// TwinCAT 3 PLC project PLC
// Title: abc
// Company: abc
// ProjectVersion: 1.0
// ProgramVersion: 3.1.0.8
// libraries:
//   Tc2_Standard, * (Beckhoff Automation GmbH)
//   Tc2_System, * (Beckhoff Automation GmbH)
//   Tc3_Interfaces, * (Beckhoff Automation GmbH)
//   Tc3_Module, * (Beckhoff Automation GmbH)
// project tree:
//   DUTs/ PLCStruct.TcDUT, TComplexStruct.TcDUT, TSimpleStruct.TcDUT (not stored)
//   GVLs/ GVL.TcGVL
//   / PlcTask.TcTTO (not stored)
//   POUs/ FB_Math.TcPOU, MAIN.TcPOU
//   Version/ Global_Version.TcGVL
// real-time tasks:
//   TASK PlcTask: cycle T#10ms, priority 20, ADS port 350

// ---- DUTs/PLCStruct.TcDUT
TYPE PLCStruct :
STRUCT
	intVal 	: INT;
  	dintVal	: DINT;
  	byteVal	: SINT;
  	lrealVal: LREAL;
  	realVal	: REAL;
END_STRUCT
END_TYPE

// ---- DUTs/TComplexStruct.TcDUT
TYPE TComplexStruct :
STRUCT
	intVal 			: INT:=1200;
	dintArr			: ARRAY[0..3] OF DINT := [1,2,3,4];
	boolVal			: BOOL := FALSE;
	byteVal			: BYTE:=10;
	stringVal 		: STRING(5) := 'hallo';
	simpleStruct1	:  TSimpleStruct;
END_STRUCT
END_TYPE

// ---- GVLs/GVL.TcGVL
VAR_GLOBAL
	//Sample21
	REAL32_1 AT %MB0 : REAL;  (* 1 *)
        REAL32_2 AT %MB4 : REAL;  (* 2 *)
        REAL32_3 AT %MB8 : REAL;  (* 3 *)
        REAL32_4 AT %MB12: REAL;  (* 4 *)
        REAL32_5 AT %MB16: REAL;  (* 5 *)

        REAL64_1 AT %MB20 : LREAL;  (* 6 *)
        REAL64_2 AT %MB28 : LREAL;  (* 7 *)
        REAL64_3 AT %MB36 : LREAL;  (* 8 *)
        REAL64_4 AT %MB44 : LREAL;  (* 9 *)
        REAL64_5 AT %MB52 : LREAL;  (* 10 *)

        INT32_1 AT %MB60 : DINT;  (* 11 *)
        INT32_2 AT %MB64 : DINT;  (* 12 *)
        INT32_3 AT %MB68 : DINT;  (* 13 *)
        INT32_4 AT %MB72 : DINT;  (* 14 *)
        INT32_5 AT %MB76 : DINT;  (* 15 *)

        UINT32_1 AT %MB80 : UDINT;  (* 16 *)
        UINT32_2 AT %MB84 : UDINT;  (* 17 *)
        UINT32_3 AT %MB88 : UDINT;  (* 18 *)
        UINT32_4 AT %MB92 : UDINT;  (* 19 *)
        UINT32_5 AT %MB96 : UDINT;  (* 20 *)

        INT16_1 AT %MB100 : INT;  (* 21 *)
        INT16_2 AT %MB102 : INT;  (* 22 *)
        INT16_3 AT %MB104 : INT;  (* 23 *)
        INT16_4 AT %MB106 : INT;  (* 24 *)
        INT16_5 AT %MB108 : INT;  (* 25 *)

        UINT16_1 AT %MB110 : UINT;  (* 26 *)
        UINT16_2 AT %MB112 : UINT;  (* 27 *)
        UINT16_3 AT %MB114 : UINT;  (* 28 *)
        UINT16_4 AT %MB116 : UINT;  (* 29 *)
        UINT16_5 AT %MB118 : UINT;  (* 30 *)

        INT8_1 AT %MB120 : SINT;  (* 31 *)
        INT8_2 AT %MB121 : SINT;  (* 32 *)
        INT8_3 AT %MB122 : SINT;  (* 33 *)
        INT8_4 AT %MB123 : SINT;  (* 34 *)
        INT8_5 AT %MB124 : SINT;  (* 35 *)

        UINT8_1 AT %MB125 : USINT;  (* 36 *)
        UINT8_2 AT %MB126 : USINT;  (* 37 *)
        UINT8_3 AT %MB128 : USINT;  (* 38 *)
        UINT8_4 AT %MB129 : USINT;  (* 39 *)
        UINT8_5 AT %MB130 : USINT;  (* 40 *)

        BOOL_1 AT %MX131.0 : BOOL;  (* 41 *)
        BOOL_2 AT %MX131.1 : BOOL;  (* 42 *)
        BOOL_3 AT %MX131.2 : BOOL;  (* 43 *)
        BOOL_4 AT %MX131.3 : BOOL;  (* 44 *)
        BOOL_5 AT %MX131.4 : BOOL;  (* 45 *)

        ARRAY_1 : ARRAY[1 .. 10] OF SINT; (* 46 *)
        ARRAY_2 : ARRAY[1 .. 10] OF INT;  (* 47 *)
        ARRAY_3 : ARRAY[1 .. 10] OF DINT; (* 48 *)
        ARRAY_4 : ARRAY[1 .. 10] OF LREAL;(* 49 *)
        ARRAY_5 : ARRAY[1 .. 10] OF BOOL; (* 50 *)

        STRING_1 : STRING(20);
END_VAR

// ---- Version/Global_Version.TcGVL
// This function has been automatically generated from the project information.
VAR_GLOBAL CONSTANT
	{attribute 'const_non_replaced'}
	stLibVersion_abc : ST_LibVersion := (iMajor := 1, iMinor := 0, iBuild := -1, iRevision := -1, sVersion := '1.0');
END_VAR

// ---- POUs/FB_Math.TcPOU
FUNCTION_BLOCK FB_Math
VAR
	calls : INT;
END_VAR

{attribute 'TcRpcEnable'}
METHOD Addition
VAR_INPUT
	a: DINT;
	b: DINT;
END_VAR
VAR_OUTPUT
	sum: DINT;
END_VAR
sum := a + b;
calls := calls + 1;
END_METHOD

END_FUNCTION_BLOCK

// ---- POUs/MAIN.TcPOU
PROGRAM MAIN
VAR
	//Sample 01 and 02
	nCounter     AT %MD0 :DWORD;
	TP_1		: TP;
	TOGGEL		: BOOL;

	//Sample03
	 boolVal   : BOOL;
	 intVal    : INT;
	 dintVal   : DINT;
	 sintVal   : SINT;
	 lrealVal  : LREAL;
	 realVal   : REAL;
	 stringVal : STRING(20);
	 
	//Sample10
	text : STRING[30] := 'Hello TwinCAT';
	
	//Sample11
	Time1:TIME := T#21H33M23S231MS;
    Date1:DT:=DT#1993-06-12-15:36:55.40;
	
	//Sample12
	PLCArray : ARRAY [0..99] OF INT;
  	Index: BYTE;
	
	//Sample13
	PLCStruct : PLCStruct;	
	
	//Sample14
	(*primitive Types*)
	bool1:BOOL := FALSE;
	int1:INT := 30000;
	dint1:DINT:=125000;
	usint1:USINT:=200;
	real1:REAL:= 1.2;
	lreal1:LREAL:=3.5;

	(*string Types*)
	str1:STRING := 'this is a test string';
	str2:STRING(5) := 'hallo';

	(*struct Types*)
	complexStruct1 : TComplexStruct;
	
	//Sample22
	uintValue 	: UDINT 	:= 54321;
	boolValue	: BOOL 		:= TRUE;
	dintValue	: DINT		:= -12345678;
	
	//Sample30
	fbMath	: FB_MATH;
	TON1: TON;
END_VAR

//Sample 01 and 02
nCounter := nCounter + 1;

//Sample 03
sintVal := sintVal + 1;
dintVal := dintVal + 5;
realVal := realVal + 0.1;
lrealVal := lrealVal + 0.1;

boolVal := FALSE;
TON1(IN:= TRUE, PT:= T#200MS, Q=> boolVal);
IF boolVal THEN
	IF intval > 12 THEN
		intval := 0;
	END_IF
	intVal := intVal + 1;
	stringVal := LEFT(Text, intVal);
	TON1(IN:= FALSE);
END_IF

//Sample12
FOR Index := 0 TO 99 DO
  PLCArray[Index] := 3500 + INDEX;
END_FOR

END_PROGRAM
